PROGRAM PRG_FactoryIO_ModbusTCP_old
// Dépendance Tc2_ModbusSrv (TF6250-Modbus-TCP)
// FB_Bool_To_Word + FB_Word_To_Bool
VAR
	fb_FactoryIO_ModbusTCP : FB_FactoryIO_ModbusTCP_Read;
END_VAR

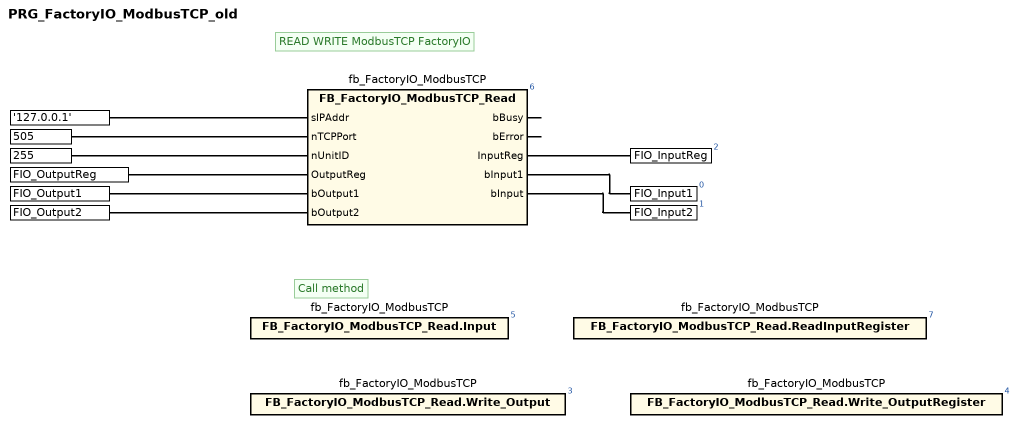
FIO_Input1 := fb_FactoryIO_ModbusTCP.bInput1;
FIO_Input2 := fb_FactoryIO_ModbusTCP.bInput;
FIO_InputReg := fb_FactoryIO_ModbusTCP.InputReg;
fb_FactoryIO_ModbusTCP.Write_Output();
fb_FactoryIO_ModbusTCP.Write_OutputRegister();
// Call method
fb_FactoryIO_ModbusTCP.Input();
// READ WRITE ModbusTCP FactoryIO
fb_FactoryIO_ModbusTCP(
    sIPAddr := '127.0.0.1',
    nTCPPort := 505,
    nUnitID := 255,
    OutputReg := FIO_OutputReg,
    bOutput1 := FIO_Output1,
    bOutput2 := FIO_Output2); // FB_FactoryIO_ModbusTCP_Read
fb_FactoryIO_ModbusTCP.ReadInputRegister();

END_PROGRAM

(* stored: Version 1.1.0.1, ProductVersion 3.1.4024.11
   POU PRG_FactoryIO_ModbusTCP_old: Id {f21e239b-c62a-4334-a832-526a3939b4fa}, SpecialFunc None *)
